// TIA Portal V20 export
DATA_BLOCK "SendFData_BA10AC1"   // DB129
// stored: InstanceOfName Safety.GM_SendFData, InstanceOfType FB, Namespace Safety
"Safety.GM_SendFData"
   // VAR_INPUT
   //    Connection_ID_Send : Word;
   //    Connection_ID_Receive : Word;
   // END_VAR
   // VAR_IN_OUT
   //    Send_Array : Array[0..121] of Byte;
   //    Receive_Ack_Send_Array : Array[0..21] of Byte;
   // END_VAR
   // VAR
   //    instTSendData : TSEND;
   //    instTSendAck { S7_SetPoint := 'True'} : TSEND;
   //    statErrorSendData { S7_SetPoint := 'True'} : Word;
   //    statErrorSendAck : Word;
   //    statSendTimer { S7_SetPoint := 'True'} : TON_TIME;
   // END_VAR
BEGIN
END_DATA_BLOCK
